Universal Robots PolyScope program: 10.08.24.urp

ProgramRoot directory=/programs/Bas; kinematics=(a=[0, -0.612, -0.5723, 0, 0, 0], d=[0.1273, 0, 0, 0.16394, 0.1157, 0.0922], alpha=[1.5708, 0, 0, 1.5708, -1.5708, 0], deltaTheta=[0, 0, 0, 0, 0, 0], status=notInitialized); name=10.08.24; programVersion=(project__name=PolyScope, major__version=1, minor__version=8, svn__revision=25319, build__date=Oct 19 2016, 16:34:22); robotEnvironmentFileName=default; serialNumberRobot=2013202566
  MainProgram cartesianAcceleration=1.2; cartesianSpeed=0.25; jointAcceleration=1.3962634015954636; jointSpeed=1.0471975511965976; moveAsFastAsPossible=true; sharedProcessMoveBlendRadius=0.025; featureReference=(installationNameReference=Base); motionType=JOINT_SPACE; runOnlyOneCycle=true
    Move cartesianAcceleration=1.2; cartesianSpeed=0.25; jointAcceleration=1.3962634015954636; jointSpeed=1.0471975511965976; moveAsFastAsPossible=true; sharedProcessMoveBlendRadius=0.025; featureReference=(installationNameReference=Base); motionType=JOINT_SPACE
      Waypoint blendRadius=0.05; cartesianAcceleration=1.2; cartesianSpeed=0.25; jointAcceleration=1.3962634015954636; jointSpeed=1.0471975511965976; nextMotionTime=2.0; stoppoint=true; useSharedBlendParameter=true; useSharedParameters=true; position=TCP in base x=111.429 y=-500.519 z=756.038 mm, rx=2.1543 ry=2.2752 rz=0.0352 rad; joints [-59.064, -72.421, -93.7, 256.221, 91.368, 117.812] deg; positionType=FIXED_POSITION; waypointPoseInFeatureCoordinates=(pos=(x=0.11142891086151867, y=-0.5005186797118292, z=0.7560383551799643), rot=(x=2.1543032046418866, y=2.275180357187861, z=0.035242037630503806)); name=Waypoint_1
    Suppressed 
    Suppressed 
    Script type=1; cachedFileContents=textmsg(get_actual_tcp_pose())
      | 
      | port = 5005
      | ip = "192.168.0.45"
      | socket_name = "fadil"
      | 
      | socket = socket_open(ip, port, socket_name)
      | movel (p[0.111428, -0.500535, 0.756028, 2.15432, 2.27516, 0.0352882])
      | sleep(0.1)
      | set_digital_out(0,True)
      | 
      | while(True):
      | socket_send_string("trig", socket_name)
      | textmsg("trig send")
      | 
      | receive = socket_read_ascii_float(2, socket_name)
      | textmsg(receive)
      | sleep(0.01)
      | 
      | #cTcp = get_actual_tcp_pose()
      | a=get_actual_tcp_pose()
      | 
      | x= receive[1] / 1000
      | y= receive[2] / 1000
      | z= 0.241219
      | 
      | movel (p[x, y, 0.35, a[3], a[4], a[5]], 0.3, 0.5)
      | movel (p[x, y, z, a[3], a[4], a[5]])
      | sleep(0.1)
      | set_digital_out(0,False)
      | movel (p[x, y, 0.590, a[3], a[4], a[5]])
      | sleep(0.1)
      | #movel (p[-0.711215, 0.0412935, 0.462286, 2.70785, 1.56442, 0.0299764])
      | #sleep(0.1)
      | #movel (p[-0.711215, 0.0412935, 0.362286, 2.70785, 1.56442, 0.0299764])
      | #sleep(0.1)
      | 
      | 
      | movel (p[x-0.111, y, 0.756028, a[3], a[4], a[5]], 0.3, 0.5)
      | sleep(0.1)
      | set_digital_out(0,True)
      | socket_send_string(get_actual_tcp_pose(), socket_name)
      | end; scriptFile=/programs/Bas/1.8.script
    Suppressed 
